PROGRAM POU_SetaEmergencia
VAR
END_VAR

(* GVL GENERAL *)

GVL_General.sBeltConveyor.bSortingCintaDistribucion := FALSE;
GVL_General.sBeltConveyor.bSortingCintaEntrada := FALSE;
GVL_General.sBeltConveyor.bSortingCintaInicial := FALSE;


GVL_General.bStopBlade1 := FALSE;


GVL_General.sBeltConveyor.bCintaAzul1 := FALSE;
GVL_General.sBeltConveyor.bCintaAzul2 := FALSE;

GVL_General.sBeltConveyor.bCintaMetal1 := FALSE;
GVL_General.sBeltConveyor.bCintaMetal2 := FALSE;

GVL_General.sBeltConveyor.bCintaVerde1 := FALSE;
GVL_General.sBeltConveyor.bCintaVerde2 := FALSE;


(* GVL ENTRADA *)

GVL_Sorting.sPusherA.Pusher := FALSE;
GVL_Sorting.sPusherV.Pusher := FALSE;
GVL_Sorting.sPusherM.Pusher := FALSE;


(* GVL GUARDADO *)

GVL_StackBox.bStopBladeA1 := FALSE;
GVL_StackBox.bStopBladeA2 := FALSE;

GVL_StackBox.bStopBladeV1 := FALSE;
GVL_StackBox.bStopBladeV2 := FALSE;

GVL_StackBox.bStopBladeM1 := FALSE;
GVL_StackBox.bStopBladeM2 := FALSE;

GVL_StackBox.sPickAndPlaceA.bGrab := FALSE;
GVL_StackBox.sPickAndPlaceA.bGripperCCW := FALSE;
GVL_StackBox.sPickAndPlaceA.bGripperCW := FALSE;
GVL_StackBox.sPickAndPlaceA.bMovementX := FALSE;
GVL_StackBox.sPickAndPlaceA.bMovementZ := FALSE;
GVL_StackBox.sPickAndPlaceA.bRotateCCW := FALSE;
GVL_StackBox.sPickAndPlaceA.bRotateCW := FALSE;

END_PROGRAM

(* stored: Version 1.1.0.1, ProductVersion 3.1.4024.12
   POU POU_SetaEmergencia: Id {673bb672-76e7-47b1-8f3a-f753faa32ba6}, SpecialFunc None *)
